{attribute 'strict'}
TYPE E_VisionResult :
(
	UNDEFINE 						:= 0,
	LESS_QTTY_CAM 					:= 10,
	LESS_QTTY_HOLE					:= 20,
	LESS_QTTY_SOUND_OUTLET			:= 30,
	STONE_STUCK_IN_HOLE				:= 40,
	WRONG_POSITION_SOUND_OUTLET		:= 50,
	SCRATCH							:= 60,
	DENT							:= 70,
	DIRT_CONTAMINATION				:= 80,
	WRONG_POSITION_CAM				:= 90,					
	DEFORM							:= 100,
	INSUFFICIENT_CHIPPING			:= 110
	//BURR							:= 120,
	
);
END_TYPE

(* stored: Version 1.1.0.1, ProductVersion 3.1.4024.9
   DUT E_VisionResult: Id {b10f470d-097d-410b-98da-d876df638217} *)
